(* PLC project CoDeSys External Library Template, WAGO e!COCKPIT e!COCKPIT, author 3S - Smart Software Solutions GmbH *)
(* stored: creationDateTime 2019-10-29T12:22:40.867242, version 3.5.5.30, modificationDateTime 2019-10-24T14:40:07.960949, organization 3S - Smart Software Solutions GmbH *)
(* Library project template with all possible element types, docu and a sample project structure *)

FUNCTION fnKomunikatDaneSzukajZmiennej : BOOL
  VAR_INPUT
    sKomunikat : alSTRINGKomunikat;
    sZmienna : STRING;
  END_VAR
  VAR
    intBlad : INT;
    typKomunikat : typKomunikat;
    intPozycja1 : INT;
    intPozycja2 : INT;
  END_VAR

            fnKomunikatInOut(	xStringNaStrukture := TRUE ,
					xStringUpdateZeStruktury := FALSE ,
					xStrukturyNaString := FALSE ,
					xWyczyscStrukture := FALSE ,
					xAktualizujZnacznikCzasu := FALSE ,
					xAktualizujDlugoscDanych := FALSE ,
					sKomunikat := sKomunikat ,
					typKomunikat := typKomunikat ,
					intBlad := intBlad);

IF FIND(typKomunikat.sDane , sZmienna) <> 0 THEN
	fnKomunikatDaneSzukajZmiennej := TRUE;
	ELSE
	fnKomunikatDaneSzukajZmiennej := FALSE;
END_IF
				
					
					
					
					
					
					
          
END_FUNCTION
